/// container for all communication data types that are used by the unit
TYPE ScriblyComRef :
STRUCT
  Publish : REFERENCE TO ScriblyComPublish; 
  Subscribe : REFERENCE TO ScriblyComSubscribe; 
END_STRUCT
END_TYPE

(* stored: Version 1.1.0.1
   DUT ScriblyComRef: Id {116198e2-1f9f-4076-b579-2ecaebbb9b30} *)
